// TIA Portal V19 export
TYPE "MES_Err"
   STRUCT
      Presence : Bool;
      Code : DInt;
      Description : String;
   END_STRUCT;
END_TYPE
